FUNCTION_BLOCK PUBLIC enable_disable_driver
VAR_INPUT
	DRIVER:INT;
	CWORD:INT;
END_VAR

IF(DRIVER=0) THEN
	GVL.robotdata.motorCword[0]:=CWORD;
	GVL.robotdata.motorCword[1]:=CWORD;
ELSIF DRIVER=1 THEN
	GVL.robotdata.motorCword[2]:=CWORD;
ELSIF DRIVER=2 THEN
	GVL.robotdata.motorCword[3]:=CWORD;
END_IF

st_command.command:=0;

END_FUNCTION_BLOCK

(* stored: Version 1.1.0.1, ProductVersion 3.1.4024.12
   POU enable_disable_driver: Id {60c35106-513c-4441-af37-097c93551c05}, SpecialFunc None *)
